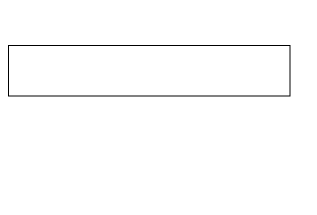
[picture p24: P60013 (HMI screen)]
rectangle at (270,210)-(321,241): text "ESC"
rectangle at (270,210)-(321,241): text "ESC"; invisible if NOT.alarm
rectangle at (20,80)-(302,131): text "Overspeed stage 2 / braking level:"
rectangle at (20,140)-(302,191): text "Overspeed stage 3 / braking level:"
rectangle at (220,90)-(301,121): text "%s %%"; shows stage2; invisible if editMode
rectangle at (220,150)-(301,181): text "%s %%"; shows stage3
rectangle at (20,40)-(302,71): text "Band brake slip level:"
rectangle at (220,40)-(301,71): text "%s %%"; shows bandSlip
*)

(* Visualisation START_PAGE/MAIN_MANU/MAIN_MENU_1/DISPLAY_SETUP/1_DISPLAY_SETUP/2_Set_Water_Brake_Limit/P60014
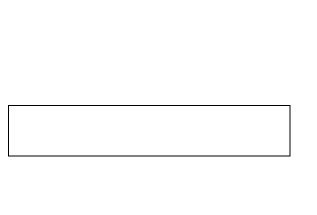
rectangle at (270,210)-(321,241): text "ESC"
rectangle at (270,210)-(321,241): text "ESC"; invisible if NOT.alarm
rectangle at (20,80)-(302,131): text "Overspeed stage 2 / braking level:"
rectangle at (20,140)-(302,191): text "Overspeed stage 3 / braking level:"
rectangle at (220,90)-(301,121): text "%s %%"; shows stage2
rectangle at (220,150)-(301,181): text "%s %%"; shows stage3; invisible if editMode
rectangle at (20,40)-(302,71): text "Band brake slip level:"
rectangle at (220,40)-(301,71): text "%s %%"; shows bandSlip
*)

(* Visualisation START_PAGE/MAIN_MANU/MAIN_MENU_1/DISPLAY_SETUP/1_DISPLAY_SETUP/Set_band_slip_level/P60015
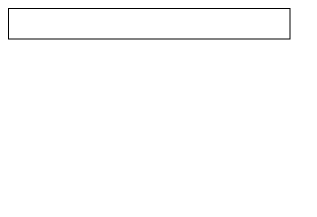
rectangle at (20,80)-(302,131): text "Overspeed stage 2 / braking level:"
rectangle at (20,140)-(302,191): text "Overspeed stage 3 / braking level:"
rectangle at (220,90)-(301,121): text "%s %%"; shows stage2
rectangle at (220,150)-(301,181): text "%s %%"; shows stage3
rectangle at (20,40)-(302,71): text "Band brake slip level:"
rectangle at (220,40)-(301,71): text "%s %%"; shows bandSlip; invisible if editMode
rectangle at (270,210)-(321,241): text "ESC"
rectangle at (270,210)-(321,241): text "ESC"; invisible if NOT.alarm
*)

(* Visualisation START_PAGE/MAIN_MANU/MAIN_MENU_1/DISPLAY_SETUP/1_DISPLAY_SETUP/P65000
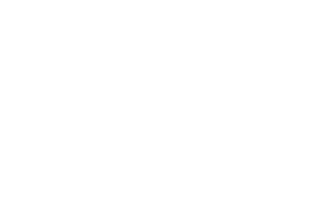
rectangle at (20,150)-(302,201): text "Overspeed stage 3 / braking level:"; alarm colour if SELECT_PAGE.MenuItem=3
rectangle at (20,90)-(302,141): text "Overspeed stage 2 / braking level:"; alarm colour if SELECT_PAGE.MenuItem=2
rectangle at (270,210)-(321,241): text "ESC"
rectangle at (270,210)-(321,241): text "ESC"; invisible if NOT.alarm
rectangle at (220,100)-(301,131): text "%s %%"; shows stage2
rectangle at (220,160)-(301,191): text "%s %%"; shows stage3
rectangle at (20,50)-(302,81): text "Band brake slip level:"; invisible if TRUE; alarm colour if SELECT_PAGE.MenuItem=1
rectangle at (220,50)-(301,81): text "%s %%"; shows bandSlip; invisible if TRUE
*)
